FUNCTION_BLOCK Fail_scenarios_HMI (* Service Interface Function Block Type *)
  (* Standard: 61499-2 *)
  (* Version 0.0, 5/14/2019, erik, nxtControl GmbH, template *)
  PACKAGE Main;
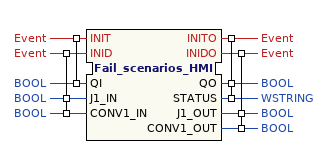
  EVENT_INPUT
    INIT WITH QI;
    INID WITH J1_IN, CONV1_IN;
  END_EVENT
  EVENT_OUTPUT
    INITO WITH QO, STATUS;
    INIDO WITH J1_OUT, CONV1_OUT;
  END_EVENT
  VAR_INPUT
    QI : BOOL;
    J1_IN : BOOL;
    CONV1_IN : BOOL;
  END_VAR
  VAR_OUTPUT
    QO : BOOL;
    STATUS : WSTRING;
    J1_OUT : BOOL;
    CONV1_OUT : BOOL;
  END_VAR
END_FUNCTION_BLOCK
